(* PLC project CoDeSys External Library Template, WAGO e!COCKPIT e!COCKPIT, author 3S - Smart Software Solutions GmbH *)
(* stored: creationDateTime 2019-10-29T12:37:19.4117826, version 3.5.5.30, modificationDateTime 2019-10-29T12:36:39.3744516, organization 3S - Smart Software Solutions GmbH *)
(* Library project template with all possible element types, docu and a sample project structure *)

(* values of enumPPPSLicznikCieplaMultical602ErrorKlasa: AlarmCzujnikaPrzeplywu: Alarm braku zmiany wartości czujnika przepływu; AlarmCzujnikaZasilania: Alarm braku zmiany wartości czujnika temp. zasilania; AlarmCzujnikaPowrotu: Alarm braku zmiany wartości czujnika temp. powrotu *)

(* Autor: Artur Wyszomirski, 2019-08-08-AWy Prawa majątkowe: Solwena Sp. z o.o., Aktualizacje: Opis: Klasy alarmów w fb licznia ciepła Multical602 *)
{attribute 'qualified_only'}
{attribute 'strict'}
TYPE enumPPPSLicznikCieplaMultical602ErrorKlasa : (BrakKomunikacji := enumKlasaAlarmu.AwariaAutomatyki, AlarmCzujnikaPrzeplywu := enumKlasaAlarmu.AwariaAutomatyki, AlarmCzujnikaZasilania := enumKlasaAlarmu.AwariaAutomatyki, AlarmCzujnikaPowrotu := enumKlasaAlarmu.Ostrzezenie);
END_TYPE
